(* IEC 61131-3 sources: PruebaSimaticAX/src, 2 files *)

(* ---- Counter.st ---- *)
USING Simatic.Ax.Conversion;
NAMESPACE Mylib

    CLASS Counter
        VAR
            Value : INT;
        END_VAR

        METHOD PUBLIC CountUp
            Value:= Value + 1;
        END_METHOD

        METHOD PUBLIC CountDown
            Value:= Value - 1;
        END_METHOD

        METHOD SetZero
            Value:= 0;
        END_METHOD

        METHOD PUBLIC GetValue :  INT
            GetValue := Value;
        END_METHOD

    END_CLASS

END_NAMESPACE

(* ---- wrapper.st ---- *)
NAMESPACE Mylib

    FUNCTION_BLOCK Wrapper

        VAR_INPUT
            CountUp : BOOL;
            CountDown : BOOL;
        END_VAR

        VAR
            CounterInstance : Counter;
        END_VAR

    IF CountUp THEN
        CounterInstance.CountUp();
    ELSIF CountDown THEN
        CounterInstance.CountDown();
    END_IF;

    END_FUNCTION_BLOCK

END_NAMESPACE
